// TIA Portal V18 export
// export: Created 2026-06-08T16:32:19.2693068Z, ExportSetting WithDefaults, DisplayName Totally Integrated Automation Portal, DisplayVersion V18, DisplayName TIA Portal Openness, DisplayVersion V18, DisplayName TIA Portal Version Control Interface, DisplayVersion V18, DisplayName STEP 7 Professional, DisplayVersion V18, DisplayName STEP 7 Safety, DisplayVersion V18, DisplayName WinCC Professional, DisplayVersion V18
VAR_GLOBAL   // PLC tag table "All_Tags"
   CCC1 AT %I10.0 : Bool;
   CCC2 AT %I10.1 : Bool;
   Tag_1 AT %M5.6 : Bool;
   Tag_2 AT %M5.7 : Bool;
   Tag_3 AT %M6.0 : Bool;
   Tag_4 AT %M6.1 : Bool;
   Tag_5 AT %M6.2 : Bool;
   Tag_6 AT %M6.3 : Bool;
   Tag_7 AT %M6.4 : Bool;
   Tag_8 AT %M6.5 : Bool;
   Tag_9 AT %M6.6 : Bool;
END_VAR
